# EPICS autosave request: iocBoot/iocImg/ccs_auto_settings.req
file "tlccs_settings.req",          P=$(P),  R=det1:
file "NDStdArrays_settings.req",    P=$(P),  R=trace1:
file "commonPlugin_settings.req",   P=$(P)
